PROGRAM MAIN
VAR
	bStart,bRun: BOOL;
	nVar1,nVar2: INT;
END_VAR

bRrun := bStart;
nVar1 :=nVar2+1;

END_PROGRAM

(* stored: Version 1.1.0.1, ProductVersion 3.1.4024.13
   POU MAIN: Id {87b87ea4-bd69-47fa-9278-a0a403183129}, SpecialFunc None *)
